FUNCTION Simula_Compila_Sta 
VAR_INPUT
	nNodo 	: UINT;	// Nodo partenza
	bCarico	: BOOL; // Stato Carico (True)
END_VAR
VAR_INPUT
 	auxSta   : REFERENCE TO STA_ASRV;
END_VAR

//--------------------------------------------------------
// Simula Compilazione Stato Inziale ASRV
// Elaborata impulsivamente  compila stato iniziale ASRV
//--------------------------------------------------------
//---------------------
// Stato inziale ASRV
//---------------------
auxSta.Pos_ASRV := nNodo;	// Nodo partenza;
auxSta.offset_da_nodo_ASRV	:=0;		
auxSta.Stato_Miss_ASRV 		:=0;
auxSta.ptr_step_ASRV		:=0;
auxSta.Perc_Batteria_ASRV	:=100;

auxSta.Stato_ASRV.In_Automatico := TRUE;
auxSta.Stato_ASRV.In_Allarme 	:= FALSE;
auxSta.Stato_ASRV.Ok_Prog		:= TRUE;
auxSta.Stato_ASRV.PosSoll_0		:= FALSE;
auxSta.Stato_ASRV.PosSoll_1		:= FALSE;
auxSta.Stato_ASRV.Carico		:= bCarico;	// Stato carico
IF bCarico = FALSE THEN
	auxSta.Peso_Teorico_ASRV	:= 0;	
END_IF 
auxSta.Stato_ASRV.Su_Nodo		:= TRUE;

END_FUNCTION

(* stored: Version 1.1.0.1, ProductVersion 3.1.4024.11
   POU Simula_Compila_Sta: Id {4399f744-729f-41ce-8336-cbd7037a9206}, SpecialFunc None *)
